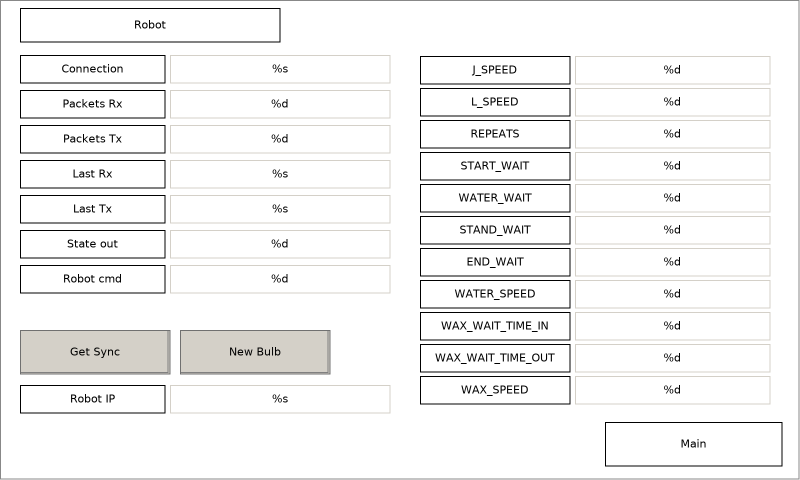
VISUALIZATION Robot  // 800x480
    Rectangle (605,422 177x44), "Main"
        OnMouseDown: change screen: Main
    Rectangle (20,8 260x34), "Robot"
    Rectangle (20,55 145x28), "Connection"
    Textfield (170,55 220x28), "%s", text variable: GVL_Robot.stRobot.sConnStateText
    Rectangle (20,90 145x28), "Packets Rx"
    Textfield (170,90 220x28), "%d", text variable: GVL_Robot.stRobot.nPacketsRx
    Rectangle (20,125 145x28), "Packets Tx"
    Textfield (170,125 220x28), "%d", text variable: GVL_Robot.stRobot.nPacketsTx
    Rectangle (20,160 145x28), "Last Rx"
    Textfield (170,160 220x28), "%s", text variable: GVL_Robot.stRobot.sLastMessage
    Rectangle (20,195 145x28), "Last Tx"
    Textfield (170,195 220x28), "%s", text variable: GVL_Robot.stRobot.sLastTxMessage
    Rectangle (20,230 145x28), "State out"
    Textfield (170,230 220x28), "%d", text variable: GVL_Robot.stParams.nStateOut
    Rectangle (20,265 145x28), "Robot cmd"
    Textfield (170,265 220x28), "%d", text variable: GVL_Robot.stParams.nRobotCmd
    Button (20,330 150x44), "Get Sync"
        tap GVL_Robot.stParams.bGetSync
    Button (180,330 150x44), "New Bulb"
        tap GVL_Robot.stParams.bTriggerNewBulb
    Textfield (575,280 195x28), "%d", text variable: GVL_Robot.stParams.WATER_SPEED
        OnMouseClick: write the text variable via Default, min 0, max 100
    Rectangle (420,56 150x28), "J_SPEED"
    Textfield (575,56 195x28), "%d", text variable: GVL_Robot.stParams.J_SPEED
        OnMouseClick: write the text variable via Default, min 1, max 100
    Rectangle (420,88 150x28), "L_SPEED"
    Textfield (575,88 195x28), "%d", text variable: GVL_Robot.stParams.L_SPEED
        OnMouseClick: write the text variable via Default, min 1, max 100
    Rectangle (420,120 150x28), "REPEATS"
    Textfield (575,120 195x28), "%d", text variable: GVL_Robot.stParams.REPEATS
        OnMouseClick: write the text variable via Default, min 1, max 10
    Rectangle (420,152 150x28), "START_WAIT"
    Textfield (575,152 195x28), "%d", text variable: GVL_Robot.stParams.START_WAIT
        OnMouseClick: write the text variable via Default, min 10, max 10000
    Rectangle (420,184 150x28), "WATER_WAIT"
    Textfield (575,184 195x28), "%d", text variable: GVL_Robot.stParams.WATER_WAIT
        OnMouseClick: write the text variable via Default, min 10, max 10000
    Rectangle (420,216 150x28), "STAND_WAIT"
    Textfield (575,216 195x28), "%d", text variable: GVL_Robot.stParams.STAND_WAIT
        OnMouseClick: write the text variable via Default, min 10, max 10000
    Rectangle (420,248 150x28), "END_WAIT"
    Textfield (575,248 195x28), "%d", text variable: GVL_Robot.stParams.END_WAIT
        OnMouseClick: write the text variable via Default, min 10, max 10000
    Rectangle (420,280 150x28), "WATER_SPEED"
    Rectangle (420,312 150x28), "WAX_WAIT_TIME_IN"
    Textfield (575,312 195x28), "%d", text variable: GVL_Robot.stParams.WAX_WAIT_TIME_IN
        OnMouseClick: write the text variable via Default, min 0, max 10000
    Rectangle (420,344 150x28), "WAX_WAIT_TIME_OUT"
    Textfield (575,344 195x28), "%d", text variable: GVL_Robot.stParams.WAX_WAIT_TIME_OUT
        OnMouseClick: write the text variable via Default, min 10, max 10000
    Rectangle (420,376 150x28), "WAX_SPEED"
    Textfield (575,376 195x28), "%d", text variable: GVL_Robot.stParams.WAX_SPEED
        OnMouseClick: write the text variable via Default, min 0, max 100
    Rectangle (20,385 145x28), "Robot IP"
    Textfield (170,385 220x28), "%s", text variable: GVL_Robot.sRobotHost
        OnMouseClick: write the text variable via Default, title Robot IP address
END_VISUALIZATION

(* stored: Version 1.1.0.1, ProductVersion 3.1.4024.16
   Visu Robot: Id {a1b2c3d4-0e5f-4a6b-9c7d-000000000102} *)
